PROGRAM PB_TestRunner
VAR
TestFramework : TestFramework;
END_VAR

TestFramework();

//UnitTests.TestRunner();

END_PROGRAM

(* stored: Version 1.1.0.1, ProductVersion 3.1.4024.11
   POU PB_TestRunner: Id {d6444dd0-a407-499b-af10-d5c873f52ae3}, SpecialFunc None *)
